(* IEC 61131-3 sources: repolevel_ST_code_completion/real_groud_truth最新/repoeval_Command1/full_result, 12 files *)

(* ---- FB_AirConComfortCommand.st ---- *)
FUNCTION_BLOCK PUBLIC FB_AirConComfortCommand IMPLEMENTS I_Command

VAR
    refAirConditioning : REFERENCE TO FB_AirConditioning;
END_VAR

METHOD PUBLIC Execute
VAR
    bIsValid : BOOL;
END_VAR

// Check if the reference to the air conditioning system is valid
bIsValid := __ISVALIDREF(refAirConditioning);

IF bIsValid THEN
    // Activate the air conditioning system
    refAirConditioning.Activate();

    // Set the air conditioning system to comfort mode with a temperature of 22.0 degrees
    refAirConditioning.SetTemperature(22.0);
END_IF
END_FUNCTION_BLOCK

(* ---- FB_AirConditioning.st ---- *)
FUNCTION_BLOCK PUBLIC FB_AirConditioning
VAR_OUTPUT
	bActive			: BOOL;
	lrTemperature	: LREAL;
END_VAR

VAR
    fbStandbyCommand : FB_AirConStandbyCommand;
    fbComfortCommand : FB_AirConComfortCommand;
END_VAR

METHOD PUBLIC Activate : BOOL
VAR_OUTPUT
    bActive : BOOL;
END_VAR
bActive := TRUE;
RETURN bActive;

METHOD PUBLIC Deactivate : BOOL
VAR_OUTPUT
    bActive : BOOL;
END_VAR
bActive := FALSE;
RETURN bActive;

METHOD PUBLIC SetTemperature : BOOL
VAR_INPUT
    lrNewTemperature : LREAL;
END_VAR
VAR_OUTPUT
    lrTemperature : LREAL;
END_VAR
lrTemperature := lrNewTemperature;
RETURN TRUE;

METHOD PUBLIC ExecuteStandbyCommand : BOOL
VAR
    bResult : BOOL;
END_VAR
fbStandbyCommand.refAirConditioning := THIS^;
bResult := fbStandbyCommand.Execute();
RETURN bResult;

METHOD PUBLIC ExecuteComfortCommand : BOOL
VAR
    bResult : BOOL;
END_VAR
fbComfortCommand.refAirConditioning := THIS^;
bResult := fbComfortCommand.Execute();
RETURN bResult;

METHOD PUBLIC GetStatus : STRING
VAR
    sStatus : STRING;
END_VAR
IF bActive THEN
    sStatus := CONCAT('Active, Temperature: ', REAL_TO_STRING(lrTemperature));
ELSE
    sStatus := 'Inactive';
END_IF
RETURN sStatus;
END_FUNCTION_BLOCK

(* ---- FB_AirConStandbyCommand.st ---- *)
FUNCTION_BLOCK PUBLIC FB_AirConStandbyCommand IMPLEMENTS I_Command

VAR
    refAirConditioning : REFERENCE TO FB_AirConditioning;
END_VAR
VAR_INPUT
    bInitRetains : BOOL; // if TRUE, the retain variables are initialized (warm start / cold start)
    bInCopyCode : BOOL;  // if TRUE, the instance afterwards gets moved into the copy code (online change)
    refNewAirConditioning : REFERENCE TO FB_AirConditioning;
END_VAR

IF (__ISVALIDREF(refNewAirConditioning)) THEN
    THIS^.refAirConditioning REF= refNewAirConditioning;
ELSE
    THIS^.refAirConditioning REF= 0;
END_IF

METHOD PUBLIC Execute : BOOL
VAR_OUTPUT
    bSuccess : BOOL;
END_VAR

IF (__ISVALIDREF(refAirConditioning)) THEN
    refAirConditioning^.bActive := FALSE; // Set air conditioning to standby mode
    bSuccess := TRUE;
ELSE
    bSuccess := FALSE; // Command failed due to invalid reference
END_IF

RETURN bSuccess;
END_FUNCTION_BLOCK

(* ---- FB_CDPlayer.st ---- *)
FUNCTION_BLOCK PUBLIC FB_CDPlayer
VAR_OUTPUT
	bPlayerActive		: BOOL;
	byVolume			: BYTE;
	byTrack				: UINT;
END_VAR

# Define the methods for the FB_CDPlayer function block

METHOD PUBLIC Start
VAR_OUTPUT
	bPlayerActive		: BOOL;
	byVolume			: BYTE;
	byTrack				: UINT;
END_VAR

bPlayerActive := TRUE;

METHOD PUBLIC Stop
VAR_OUTPUT
	bPlayerActive		: BOOL;
	byVolume			: BYTE;
	byTrack				: UINT;
END_VAR

bPlayerActive := FALSE;

METHOD PUBLIC SetTrack : BOOL
VAR_INPUT
	byNewTrack			: UINT;
END_VAR
VAR_OUTPUT
	bPlayerActive		: BOOL;
	byVolume			: BYTE;
	byTrack				: UINT;
END_VAR

byTrack := byNewTrack;

METHOD PUBLIC SetVolume : BOOL
VAR_INPUT
	byNewVolume			: BYTE;
END_VAR
VAR_OUTPUT
	bPlayerActive		: BOOL;
	byVolume			: BYTE;
	byTrack				: UINT;
END_VAR

byVolume := byNewVolume;

# The FB_CDPlayer function block now includes methods to start, stop, set the track, and set the volume.
END_FUNCTION_BLOCK

(* ---- FB_Lamp.st ---- *)
FUNCTION_BLOCK PUBLIC FB_Lamp
VAR_OUTPUT
	byLevel			: BYTE;
END_VAR

VAR_INPUT
	byNewLevel		: BYTE;
END_VAR

METHOD PUBLIC SetLevel : BOOL
VAR_OUTPUT
	byLevel			: BYTE;
END_VAR
VAR_INPUT
	byNewLevel		: BYTE;
END_VAR

// Implementation of the SetLevel method
byLevel := byNewLevel;
RETURN TRUE;

// Additional functionality for FB_Lamp
METHOD PUBLIC GetLevel : BYTE
// This method returns the current level of the lamp
RETURN byLevel;

METHOD PUBLIC IsOn : BOOL
// This method checks if the lamp is on (level > 0)
IF byLevel > 0 THEN
	RETURN TRUE;
ELSE
	RETURN FALSE;
END_IF;
END_FUNCTION_BLOCK

(* ---- FB_LampSetLevelCommand.st ---- *)
FUNCTION_BLOCK PUBLIC FB_LampSetLevelCommand IMPLEMENTS I_Command

VAR
    refLamp : REFERENCE TO FB_Lamp;
    byNewLevel : BYTE;
END_VAR

METHOD PUBLIC Execute : BOOL
VAR_OUTPUT
    bSuccess : BOOL;
END_VAR

bSuccess := FALSE;

IF (__ISVALIDREF(refLamp)) THEN
    refLamp.SetLevel(byNewLevel);
    bSuccess := TRUE;
END_IF

RETURN bSuccess;
END_FUNCTION_BLOCK

(* ---- FB_MusicPlayCommand.st ---- *)
FUNCTION_BLOCK PUBLIC FB_MusicPlayCommand IMPLEMENTS I_Command

VAR
    refCDPlayer : REFERENCE TO FB_CDPlayer;
END_VAR

METHOD Execute
VAR
    refCDPlayer : REFERENCE TO FB_CDPlayer;
END_VAR

IF (__ISVALIDREF(THIS^.refCDPlayer)) THEN
    THIS^.refCDPlayer.SetVolume(40);
    THIS^.refCDPlayer.SetTrack(1);
    THIS^.refCDPlayer.Start();
END_IF
END_FUNCTION_BLOCK

(* ---- FB_MusicStopCommand.st ---- *)
FUNCTION_BLOCK PUBLIC FB_MusicStopCommand IMPLEMENTS I_Command

VAR
    refCDPlayer : REFERENCE TO FB_CDPlayer;
END_VAR

METHOD Execute
VAR
    refCDPlayer : REFERENCE TO FB_CDPlayer;
END_VAR

IF (__ISVALIDREF(THIS^.refCDPlayer)) THEN
    THIS^.refCDPlayer.Stop();
END_IF
END_FUNCTION_BLOCK

(* ---- FB_Socket.st ---- *)
FUNCTION_BLOCK PUBLIC FB_Socket
VAR_OUTPUT
	bActive		: BOOL;
END_VAR

METHOD PUBLIC On
VAR_OUTPUT
	bActive : BOOL;
END_VAR

// Set the socket to active
bActive := TRUE;

METHOD PUBLIC Off
VAR_OUTPUT
	bActive : BOOL;
END_VAR

// Set the socket to inactive
bActive := FALSE;

FUNCTION_BLOCK PUBLIC FB_SocketOnCommand IMPLEMENTS I_Command
VAR
	refSocket : REFERENCE TO FB_Socket;
END_VAR

METHOD PUBLIC Execute
// Turn the socket on by calling the On method
refSocket.On();

FUNCTION_BLOCK PUBLIC FB_SocketOffCommand IMPLEMENTS I_Command
VAR
	refSocket : REFERENCE TO FB_Socket;
END_VAR

METHOD PUBLIC Execute
// Turn the socket off by calling the Off method
refSocket.Off();

FUNCTION_BLOCK PUBLIC FB_Lamp
VAR_OUTPUT
	byLevel : BYTE; // Represents the brightness level of the lamp
END_VAR

METHOD PUBLIC SetLevel
VAR_INPUT
	iLevel : BYTE; // Input level to set the lamp brightness
END_VAR

// Set the brightness level of the lamp
byLevel := iLevel;

METHOD PUBLIC GetLevel
VAR_OUTPUT
	byLevel : BYTE; // Output the current brightness level
END_VAR

// Return the current brightness level
byLevel := byLevel;
END_FUNCTION_BLOCK

(* ---- FB_SocketOffCommand.st ---- *)
FUNCTION_BLOCK PUBLIC FB_SocketOffCommand IMPLEMENTS I_Command

VAR
    refSocket : REFERENCE TO FB_Socket;
END_VAR

METHOD PUBLIC Execute
VAR
    bSuccess : BOOL;
END_VAR
IF (__ISVALIDREF(THIS^.refSocket)) THEN
    THIS^.refSocket.Off();
    bSuccess := TRUE;
ELSE
    bSuccess := FALSE;
END_IF
RETURN bSuccess;

METHOD PUBLIC FB_init
VAR_INPUT
    bInitRetains : BOOL; // if TRUE, the retain variables are initialized (warm start / cold start)
    bInCopyCode : BOOL;  // if TRUE, the instance afterwards gets moved into the copy code (online change)
    refNewSocket : REFERENCE TO FB_Socket;
END_VAR
IF (__ISVALIDREF(refNewSocket)) THEN
    THIS^.refSocket REF= refNewSocket;
ELSE
    THIS^.refSocket REF= 0;
END_IF
END_FUNCTION_BLOCK

(* ---- FB_SocketOnCommand.st ---- *)
FUNCTION_BLOCK PUBLIC FB_SocketOnCommand IMPLEMENTS I_Command

VAR
    refSocket : REFERENCE TO FB_Socket;
END_VAR

METHOD Execute
VAR
    refSocket : REFERENCE TO FB_Socket;
END_VAR
IF (__ISVALIDREF(THIS^.refSocket)) THEN
    THIS^.refSocket.On();
END_IF
END_FUNCTION_BLOCK

(* ---- FB_SwitchPanel.st ---- *)
FUNCTION_BLOCK PUBLIC FB_SwitchPanel
VAR_INPUT
	arrSwitch		: ARRAY[1..8] OF BOOL;
END_VAR

VAR
	aiCommand		: ARRAY[1..8] OF I_Command;
	arrRtrig		: ARRAY[1..8] OF R_TRIG;
	nIndex			: INT;
END_VAR

METHOD PUBLIC FB_init : BOOL
VAR_INPUT
	bInitRetains	: BOOL; // if TRUE, the retain variables are initialized (warm start / cold start)
	bInCopyCode		: BOOL; // if TRUE, the instance afterwards gets moved into the copy code (online change)
END_VAR

VAR
	nIndex			: INT;
END_VAR

FOR nIndex := 1 TO 8 DO
	aiCommand[nIndex] := 0;
END_FOR

RETURN TRUE;

METHOD PUBLIC SetCommand : BOOL
VAR_INPUT
	nPosition		: INT;
	iCommand		: I_Command;
END_VAR

IF ((nPosition >= 1) AND (nPosition <= 8) AND (iCommand <> 0)) THEN
	aiCommand[nPosition] := iCommand;
	RETURN TRUE;
ELSE
	RETURN FALSE;
END_IF

METHOD PUBLIC ExecuteCommands : BOOL
VAR
	nIndex			: INT;
END_VAR

FOR nIndex := 1 TO 8 DO
	IF arrSwitch[nIndex] THEN
		IF aiCommand[nIndex] <> 0 THEN
			aiCommand[nIndex](); // Execute the command
		END_IF
	END_IF
END_FOR

RETURN TRUE;

METHOD PUBLIC ResetCommands : BOOL
VAR
	nIndex			: INT;
END_VAR

FOR nIndex := 1 TO 8 DO
	aiCommand[nIndex] := 0;
END_FOR

RETURN TRUE;
END_FUNCTION_BLOCK
